Fanuc KAREL source: KCL.kl

PROGRAM T
%NOLOCKGROUP
VAR
 v0 : STRING[40]
 v1 : INTEGER
BEGIN
 KCL(v0, v1)
END T
